Staubli VAL3: onStop.pgx

public program onStop(string& x_sItem[])
begin
  aioSet(io:MbAO_aMoveDis,0)
  aioSet(io:MbAO_b7Axis,0)
  logMsg("7")
end
